{attribute 'global_init_slot' := '49991'}
{attribute 'qualified_only'}
VAR_GLOBAL CONSTANT
	// filter cut-off frequency for velocity and torque
	g_curJntVelLpfCutoffFreq :LREAL := 30;
	g_cmdJntTrqLpfCutoffFreq :LREAL := 300;
	g_curJntTrqLpfCutoffFreq :LREAL := 300;
	
	// master arm joint position controller parameters
	g_posKp :ARRAY[1..g_setupJntNum] OF LREAL :=[0.0, 0.0, 0.0, 0.0, 2000];
	g_posKd :ARRAY[1..g_setupJntNum] OF LREAL :=[0.0, 0.0, 0.0, 0.0, 200 ];
	g_posKi :ARRAY[1..g_setupJntNum] OF LREAL :=[0.0, 0.0, 0.0, 0.0, 5000];
	g_posKiLimit :ARRAY[1..g_setupJntNum] OF LREAL :=[0.0, 0.0, 0.0, 0.0, 2000];// define in current
	g_posCtrlLimit :ARRAY[1..g_setupJntNum] OF LREAL :=[0.0, 0.0, 0.0, 0.0, 5000];// define in current
	
END_VAR

(* stored: Version 1.1.0.1, ProductVersion 3.1.4024.11
   GVL GVL_SetupControlParameters: Id {2ac57dba-e9b4-4856-a882-cc0b28d9a90f} *)
